FUNCTION_BLOCK JsonResponseBuilder IMPLEMENTS I_JsonResponseBuilder
VAR
	jsonDocument : FB_JsonSaxWriter;
	jsonLanguagePack : I_JsonLanguagePack;
END_VAR

METHOD AddKey
VAR_INPUT
	Key : T_MAXSTRING;
END_VAR
jsonDocument.AddKey(Key);
END_METHOD

METHOD PUBLIC AddKeyBase64
VAR_INPUT
	Key : T_MAXSTRING;
	pByte : POINTER TO BYTE;
	Size : DINT;
END_VAR
jsonDocument.AddBase64(pByte, Size);
END_METHOD

METHOD PUBLIC AddKeyBool
VAR_INPUT
	Key : T_MAXSTRING;
	Value : BOOL;
END_VAR
jsonDocument.AddKeyBool(Key, Value);
END_METHOD

METHOD PUBLIC AddKeyData
VAR_INPUT
	Key : T_MAXSTRING;
	Source : I_DataAccess;
END_VAR
VAR
	jsonSize : UDINT;
	pJsonString : POINTER TO STRING;
END_VAR
jsonSize := jsonLanguagePack.DataToJsonStringSize(Source);
pJsonString := __NEW(BYTE, jsonSize);

jsonLanguagePack.DataToJsonString(Source,pJsonString,jsonSize);

jsonDocument.AddKey(Key);
jsonDocument.AddRawObject(pJsonString^);

__DELETE(pJsonString);
END_METHOD

METHOD PUBLIC AddKeyDateTime
VAR_INPUT
	Key : T_MAXSTRING;
	Value : DATE_AND_TIME;
END_VAR
jsonDocument.AddKeyDateTime(Key, Value);
END_METHOD

METHOD PUBLIC AddKeyDcTime
VAR_INPUT
	Key : T_MAXSTRING;
	Value : DCTIME;
END_VAR
jsonDocument.AddKeyDcTime(Key, Value);
END_METHOD

METHOD PUBLIC AddKeyDint
VAR_INPUT
	Key : T_MAXSTRING;
	Value : DINT;
END_VAR
jsonDocument.AddDint(Value);
END_METHOD

METHOD PUBLIC AddKeyFileTime
VAR_INPUT
	Key : T_MAXSTRING;
	Value : FILETIME;
END_VAR
jsonDocument.AddKeyFileTime(Key, Value);
END_METHOD

METHOD PUBLIC AddKeyHexBinary
VAR_INPUT
	Key : T_MAXSTRING;
	SourceAddress : POINTER TO BYTE;
	SourceSize : DINT;
END_VAR
jsonDocument.AddHexBinary(SourceAddress,SourceSize);
END_METHOD

METHOD PUBLIC AddKeyLint
VAR_INPUT
	Key : T_MAXSTRING;
	Value : LINT;
END_VAR
jsonDocument.AddLint(Value);
END_METHOD

METHOD PUBLIC AddKeyLongString
VAR_INPUT
	Key : T_MAXSTRING;
	pString : POINTER TO STRING;
END_VAR
jsonDocument.AddKeyString(Key, pString^);
END_METHOD

METHOD PUBLIC AddKeyLreal
VAR_INPUT
	Key : T_MAXSTRING;
	Value : LREAL;
END_VAR
jsonDocument.AddKeyLreal(Key,Value);
END_METHOD

METHOD PUBLIC AddKeyNull
VAR_INPUT
	Key : T_MAXSTRING;
END_VAR
jsonDocument.AddKeyNull(Key);
END_METHOD

METHOD PUBLIC AddKeyNumber
VAR_INPUT
	Key : T_MAXSTRING;
	Value : DINT;
END_VAR
jsonDocument.AddKeyNumber(Key,Value);
END_METHOD

METHOD PUBLIC AddKeyRawArray
VAR_INPUT
	Key : T_MAXSTRING;
	Json : POINTER TO STRING;
END_VAR
jsonDocument.AddRawArray(Json^);
END_METHOD

METHOD PUBLIC AddKeyRawObject
VAR_INPUT
	Key : T_MAXSTRING;
	Json : POINTER TO STRING;
END_VAR
jsonDocument.AddRawObject(Json^);
END_METHOD

METHOD PUBLIC AddKeyReal
VAR_INPUT
	Key : T_MAXSTRING;
	Value : REAL;
END_VAR
jsonDocument.AddReal(Value);
END_METHOD

METHOD PUBLIC AddKeyString
VAR_INPUT
	Key : T_MAXSTRING;
	Value : T_MAXSTRING;
END_VAR
jsonDocument.AddKeyString(Key,Value);
END_METHOD

METHOD PUBLIC AddKeyUdint
VAR_INPUT
	Key : T_MAXSTRING;
	Value : UDINT;
END_VAR
jsonDocument.AddUdint(Value);
END_METHOD

METHOD PUBLIC AddKeyUlint
VAR_INPUT
	Key : T_MAXSTRING;
	Value : ULINT;
END_VAR
jsonDocument.AddUlint(Value);
END_METHOD

METHOD PUBLIC CopyJsonDocument : UDINT
VAR_INPUT
	pString : POINTER TO STRING;
	Size : UDINT;
END_VAR
CopyJsonDocument := jsonDocument.CopyDocument(pString^, Size);
END_METHOD

METHOD EndArray
VAR_INPUT
END_VAR
jsonDocument.EndArray();
END_METHOD

METHOD PUBLIC EndObject
jsonDocument.EndObject();
END_METHOD

METHOD FB_exit : BOOL
VAR_INPUT
	bInCopyCode : BOOL; // if TRUE, the exit method is called for exiting an instance that is copied afterwards (online change).
END_VAR
IF bInCopyCode THEN
	RETURN;
END_IF

jsonDocument.ResetDocument();
END_METHOD

METHOD FB_init : BOOL
VAR_INPUT
	bInitRetains : BOOL; // if TRUE, the retain variables are initialized (warm start / cold start)
	bInCopyCode : BOOL;  // if TRUE, the instance afterwards gets moved into the copy code (online change)
	JsonLanguagePack : I_JsonLanguagePack;
END_VAR
THIS^.jsonLanguagePack := JsonLanguagePack;
jsonDocument.ResetDocument();
END_METHOD

METHOD PUBLIC GetJsonDocument : T_MAXSTRING
VAR_INPUT
END_VAR
GetJsonDocument := jsonDocument.GetDocument();
END_METHOD

METHOD PUBLIC GetJsonDocumentLength : UDINT
VAR_INPUT
END_VAR
GetJsonDocumentLength := jsonDocument.GetDocumentLength();
END_METHOD

METHOD PUBLIC ResetDocument
VAR_INPUT
END_VAR
jsonDocument.ResetDocument();
END_METHOD

METHOD PUBLIC StartArray
jsonDocument.StartArray();
END_METHOD

METHOD PUBLIC StartObject
jsonDocument.StartObject();
END_METHOD

END_FUNCTION_BLOCK

(* stored: Version 1.1.0.1, ProductVersion 3.1.4024.12
   POU JsonResponseBuilder: Id {37120b21-9971-0f50-247e-7d64927ad18a}, SpecialFunc None
   Folder Constructor: Id {47a40186-257a-0a46-05b8-be1d43fd63e1}
   Folder Destructor: Id {f15000f6-c0d2-0d37-11db-4460700295a0}
   Method AddKey: Id {70c16e7d-b2a7-0e2e-3f8d-cb5d66b9b6f3}
   Method AddKeyBase64: Id {b3760c5f-76da-0708-31be-7fdfa3a46c91}
   Method AddKeyBool: Id {720fe712-f78b-0f1b-02d6-bb57cf0e2c63}
   Method AddKeyData: Id {12092a59-8720-036a-324e-b8fa5e7c7add}
   Method AddKeyDateTime: Id {ccec046b-2895-0ef4-0e80-e944cbbcbb4a}
   Method AddKeyDcTime: Id {35cf1758-5c0e-0d2d-2468-200be963e129}
   Method AddKeyDint: Id {ed23705b-ea3d-0628-0ed4-f9e96d008d7c}
   Method AddKeyFileTime: Id {5e967a9d-316e-0093-0623-19ff4b7a8b65}
   Method AddKeyHexBinary: Id {7acf6dcc-de88-0e76-27dd-ab7798498248}
   Method AddKeyLint: Id {2a50eb79-32e0-0f48-236b-6bf346869465}
   Method AddKeyLongString: Id {e044c8f1-a08b-0210-30f1-9b139f5da117}
   Method AddKeyLreal: Id {1e5ac397-bb46-07a0-09e5-9e2e5226be9e}
   Method AddKeyNull: Id {089daacf-1aa7-07f9-1dd5-2ce9c6901c96}
   Method AddKeyNumber: Id {4aeed987-2aad-02c4-328f-7f145201fc25}
   Method AddKeyRawArray: Id {1530986b-96fe-053c-34a4-1b6efb109207}
   Method AddKeyRawObject: Id {ff0db330-b82a-0571-0e5c-5394dcb7df62}
   Method AddKeyReal: Id {5b1ec8cc-be01-0333-2db8-7ab44b76d8e4}
   Method AddKeyString: Id {c42488da-e1ff-0be7-2529-e669d0672682}
   Method AddKeyUdint: Id {2c23f844-d9ad-0028-2183-65d75a8d24be}
   Method AddKeyUlint: Id {06c2ff7c-acce-0353-0ff0-a925965c09de}
   Method CopyJsonDocument: Id {9597d807-33a3-02b8-0851-eabbc017fbac}
   Method EndArray: Id {b607d068-f79b-0482-206b-f6092631fde3}
   Method EndObject: Id {145538db-d6e1-0ca3-2d69-99d4c9f02729}
   Method FB_exit: Id {6e890f69-4718-0598-11d7-c4113cd0b759}
   Method FB_init: Id {993dc4c1-617b-0a38-3426-c49f4f0361e8}
   Method GetJsonDocument: Id {d23f746c-5176-07aa-1d8a-15141b640c77}
   Method GetJsonDocumentLength: Id {382ab54b-7a8a-040c-0c99-8f84ef9f7e87}
   Method ResetDocument: Id {83bcf7b4-7b88-099f-2ab1-e6fd6f2c812c}
   Method StartArray: Id {f090f5a4-4a15-0d9a-3557-51f2fa4ea008}
   Method StartObject: Id {50aef9ca-0946-06be-352f-6c0daadabf43} *)
